// TIA Portal project "Proyecto_Dosificador_Mezclador_Automatico" (V17)

(* hardware
DEVICE "S7-1200 station_1"  S7-1200 Station
   slot 0: "Rack_0"  S7-1200 Rack  Rack  V1.0
   slot 1: "PLC_1"  CPU 1215C DC/DC/DC  6ES7 215-1AG40-0XB0  V4.5
*)

// ===== PLC "PLC_1"  CPU 1215C DC/DC/DC =====

VAR_GLOBAL   // PLC tag table "Entradas"
   "Sel Func" AT %I0.0 : Bool;
   "P Marcha NO" AT %I0.1 : Bool;
   "P Paro NC" AT %I0.2 : Bool;
   "P Emergencia NC" AT %I0.3 : Bool;
   "P Rearme NO" AT %I0.4 : Bool;
   "S Nivel Bajo A NO" AT %I0.5 : Bool;
   "S Nivel Bajo B NO" AT %I0.6 : Bool;
   "S Mezclador Nivel Bajo NO" AT %I0.7 : Bool;
   "S Briquetas NO" AT %I1.0 : Bool;
   "S FC Pivotante Arriba NC" AT %I1.1 : Bool;
   "S FC Pivotante Abajo NC" AT %I1.2 : Bool;
   "GM Cinta NC" AT %I1.3 : Bool;
   "GM Agitador NC" AT %I1.4 : Bool;
   "GM Pivotante NC" AT %I1.5 : Bool;
   "S Peso" AT %IW64 : Word;
END_VAR

VAR_GLOBAL   // PLC tag table "Salidas"
   "EV A Monoestable NC" AT %I1.6 : Bool;
   "EV B Monoestable NC" AT %I1.7 : Bool;
   "EV C Monoestable NC" AT %I2.0 : Bool;
   "M Cinta" AT %I2.1 : Bool;
   "M Agitador" AT %I2.2 : Bool;
   "M Pivotante Subir" AT %I2.3 : Bool;
   "M Pivotante Bajar" AT %I2.4 : Bool;
END_VAR

VAR_GLOBAL   // PLC tag table "Marcas Generales"
   "S Peso Normalizado" AT %MD2000 : Real;
   "S Peso Escalado" AT %MD2004 : Real;
   "Marca Marcha NO" AT %M2008.0 : Bool;
   "Marca Paro NC" AT %M2008.1 : Bool;
   "Marca Seguridad NC" AT %M2008.2 : Bool;
   "Marca Rearme NO" AT %M2008.3 : Bool;
   "Marca Sel Func" AT %M2008.4 : Bool;
END_VAR

ORGANIZATION_BLOCK "Main"   // OB1, LAD, ProgramCycle
TITLE = "Main Program Sweep (Cycle)"
{ S7_Optimized_Access := 'TRUE' }
VERSION : 0.1
   VAR_INPUT
      Initial_Call : Bool;   // Initial call of this OB
      Remanence : Bool;   // =True, if remanent data are available
   END_VAR
BEGIN

REGION Network 1
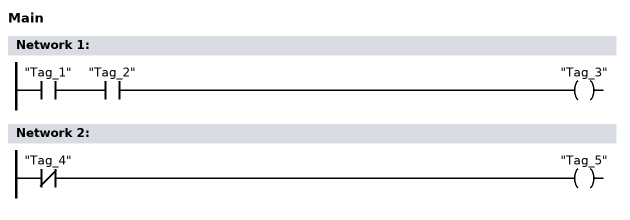
   RUNG wire#powerrail
      Contact( "Tag_1" )
      Contact( "Tag_2" )
      Coil( "Tag_3" )
   END_RUNG
   // the same network as SCL:
   "Tag_3" := "Tag_1" AND "Tag_2";
END_REGION

REGION Network 2
   RUNG wire#powerrail
      I_Contact( "Tag_4" )
      Coil( "Tag_5" )
   END_RUNG
   // the same network as SCL:
   "Tag_5" := NOT "Tag_4";
END_REGION
END_ORGANIZATION_BLOCK